// Mitsubishi GX Works2 project: group_35_Final   PLC: FX3G

// global labels: Global1
VAR_GLOBAL
  switch_check_start AT X007 : BOOL;
  cream AT D1100 : REAL;
END_VAR
VAR_GLOBAL CONSTANT
  con_false : BOOL := TRUE;
END_VAR
VAR_GLOBAL
  pulse_before_active AT X007 : BOOL;
  shity_pulse AT X011 : BOOL;
  chocolate AT D1200 : REAL;
END_VAR
VAR_GLOBAL CONSTANT
  con_chocolate : REAL := 240;
END_VAR
VAR_GLOBAL
  shity_pulse2 AT X007 : BOOL;
  shity_pulse1 AT X007 : BOOL;
  biscuit : BOOL;
END_VAR
VAR_GLOBAL CONSTANT
  con_biscuit : REAL := 6;
END_VAR
VAR_GLOBAL
  cream_input AT D1100 : REAL;
  lamp AT M2 : BOOL;
END_VAR
VAR_GLOBAL CONSTANT
  con300 : WORD := 400;
END_VAR
VAR_GLOBAL
  chocolate_input AT D1200 : REAL;
  biscit_inputnew AT D1300 : REAL;
END_VAR
VAR_GLOBAL CONSTANT
  constant6 : REAL := 6;
  contant240 : REAL := 240;
END_VAR
VAR_GLOBAL
  lamp_able_startDay AT Y002 : BOOL;
  ziluf_container : REAL;
  indicator_level1 AT Y001 : BOOL;
  kaki AT Y010 : BOOL;
  can_startday AT Y002 : BOOL;
  level1isgood AT Y001 : BOOL;
  level1done AT M2 : BOOL;
  zilufison AT X011 : BOOL;
  clockon AT TC0 : BOOL;
END_VAR
VAR_GLOBAL CONSTANT
  FourSec : REAL := 4;
  Fourcheck : WORD := 400;
END_VAR
VAR_GLOBAL
  Timer_Finish AT TS0 : BOOL;
  end_timer1 AT TS3 : BOOL;
  lamP1 AT Y005 : BOOL;
  Helo_Lamp AT M0 : BOOL;
END_VAR
VAR_GLOBAL CONSTANT
  Four_sec : INT := 40;
END_VAR
VAR_GLOBAL
  Timer_1 AT TC3 : BOOL;
END_VAR
VAR_GLOBAL CONSTANT
  One_sec : INT := 10;
END_VAR
VAR_GLOBAL
  Not_sufficnt_stuff AT M1 : BOOL;
  level1end AT Y006 : BOOL;
  lamp_2 AT Y001 : BOOL;
  Timer_2 AT TC4 : BOOL;
  TS300 : BOOL;
  end_Timer2 AT TS4 : BOOL;
  lamp_1 AT Y001 : BOOL;
  lamp0 AT Y000 : BOOL;
  Hiv_Huv_counter AT TC2 : BOOL;
  Hiv_Off AT TS2 : BOOL;
  lamp_10 AT Y001 : BOOL;
  lamp_6 AT Y006 : BOOL;
  lamp6 AT M6 : BOOL;
  Turn_on_mecA AT X010 : BOOL;
  plate_is_here AT X001 : BOOL;
  zilof_working AT Y004 : BOOL;
  high_sens AT X002 : BOOL;
  cam_sens AT X004 : BOOL;
  ziluf_lamp AT Y004 : BOOL;
  low_sens AT X003 : BOOL;
  biscuit_input : REAL;
END_VAR
VAR_GLOBAL CONSTANT
  con0 : REAL;
END_VAR
VAR_GLOBAL
  end_ziluf_lamp AT M12 : BOOL;
  qualtiy_check AT X006 : BOOL;
  analog_input AT D8280 : INT;
END_VAR
VAR_GLOBAL CONSTANT
  cons_400 : WORD := 400;
END_VAR
VAR_GLOBAL
  correct_analog AT D1111 : INT;
END_VAR
VAR_GLOBAL CONSTANT
  cons_5 : INT := 5;
END_VAR
VAR_GLOBAL
  what_is_it AT M12 : BOOL;
  yes AT M12 : BOOL;
  No AT M12 : BOOL;
END_VAR
VAR_GLOBAL CONSTANT
  cons_240 : REAL := 240;
END_VAR
VAR_GLOBAL
  con_chooclate : REAL;
END_VAR
VAR_GLOBAL CONSTANT
  cons_120 : REAL := 120;
  con400 : INT := 400;
  con300ww : REAL := 300;
END_VAR
VAR_GLOBAL
  Tvila_container : REAL;
  Tvila_timmer AT TC5 : BOOL;
END_VAR
VAR_GLOBAL CONSTANT
  tree_sec : INT := 50;
END_VAR
VAR_GLOBAL
  stop_tvila AT TS5 : BOOL;
  lamp3_off AT Y003 : BOOL;
END_VAR
VAR_GLOBAL CONSTANT
  Five_sec : INT := 50;
END_VAR
VAR_GLOBAL
  dayison AT Y007 : BOOL;
  day_is_on AT M0 : BOOL;
  lamp7 AT Y007 : BOOL;
  finish_packing AT Y002 : BOOL;
  switch_x0 AT X000 : BOOL;
  cc0_press5 AT CC0 : BOOL;
END_VAR
VAR_GLOBAL CONSTANT
  count_5 : WORD := K5;
END_VAR
VAR_GLOBAL
  switch_end_count AT CS13 : BOOL;
  m2_stop_light AT Y002 : BOOL;
  Reset_count AT Y002 : BOOL;
  Light_Y2 AT Y002 : BOOL;
  Fin6 AT Y002 : BOOL;
  Finished AT D1400 : REAL;
  count_6 AT K6 : INT;
  Stored AT D1400 : INT;
END_VAR
VAR_GLOBAL CONSTANT
  const_6 : REAL := 40;
END_VAR
VAR_GLOBAL
  Ana_Dozens AT D8282 : INT;
  ValueForOutput : REAL;
  analog_ouput AT D8282 : REAL;
  analog_output82 AT D8282 : INT;
  HELP_OUTPUT AT Y011 : BOOL;
  M_11 AT M11 : BOOL;
END_VAR
VAR_GLOBAL CONSTANT
  con_crembo6 : REAL := 6;
END_VAR
VAR_GLOBAL
  HELP_lamp_endPack AT M11 : BOOL;
END_VAR
VAR_GLOBAL CONSTANT
  con_40 : REAL := 40;
END_VAR
VAR_GLOBAL
  help_end_output AT M12 : BOOL;
  Finished_crembo AT D4000 : REAL;
  M23_finishedCH AT M23 : BOOL;
  CC13_press6 AT CC13 : BOOL;
  coub AT K6 : INT;
  M21_finish6 AT M21 : BOOL;
  press_5_finish AT CS0 : BOOL;
  press6_finished AT CS13 : BOOL;
  Restarter AT CC0 : BOOL;
  Restarter13 AT CC13 : BOOL;
  CC10_press6 AT CC10 : BOOL;
  reset0 AT CC0 : BOOL;
  reset13 AT CC13 : BOOL;
  finish_creambo AT CS13 : BOOL;
  Push_to_Spray AT X005 : BOOL;
  Sen_Full AT X004 : BOOL;
  Sen_plate AT X003 : BOOL;
  Spray AT TC6 : BOOL;
END_VAR
VAR_GLOBAL CONSTANT
  count_5sec : INT := K50;
END_VAR
VAR_GLOBAL
  Spray_light AT Y000 : BOOL;
  Spray_Timer AT TS6 : BOOL;
  HelpNOGelem AT M34 : BOOL;
  TimerEndDay AT TC9 : BOOL;
  EndDay3min AT K30 : INT;
  stop_blinking AT TS57 : BOOL;
  HELP_lamp_endday AT M5 : BOOL;
  yesGelem AT M19 : BOOL;
  finishGelem AT Y002 : BOOL;
  finishGelemCounter AT CC6 : BOOL;
END_VAR
VAR_GLOBAL CONSTANT
  count_6_finish : INT := 6;
END_VAR
VAR_GLOBAL
  finish_itertion AT Y002 : BOOL;
END_VAR
VAR_GLOBAL CONSTANT
  EndDay3sec : INT := 30;
END_VAR
VAR_GLOBAL
  TS_57 AT TS57 : BOOL;
  lamp_blinking1 AT M2 : BOOL;
  stop_blink_lamp AT M8 : BOOL;
  lamp_blinking2 AT M9 : BOOL;
  TS_7 AT TS7 : BOOL;
  TC_7 AT TS7 : BOOL;
  TC_8 AT TC8 : BOOL;
  TS_8 AT TS8 : BOOL;
  lamp_timer AT TC8 : BOOL;
  lamp_timer7 AT TC7 : BOOL;
  lamp_timer8 AT TC8 : BOOL;
  lt8 AT TS8 : BOOL;
  lt_7 AT TS7 : BOOL;
  end_lamp AT TS9 : BOOL;
  chocolate_container AT D1201 : REAL;
  biscuit_container AT D1301 : REAL;
  cream_container AT D1101 : REAL;
  Shut_Down_ziluf AT X005 : BOOL;
  Next_phase3 AT M12 : BOOL;
  lamp12 AT M120 : BOOL;
  Next_phase4 AT M120 : BOOL;
END_VAR

// task Task_01 (event TRUE, interval 0, priority 31): POU_01

PROGRAM POU_01
VAR CONSTANT
  con_cream : REAL := 300;
  con6 : REAL := 6;
END_VAR
VAR
  TC100 : BOOL;
  cam : BOOL;
END_VAR
(* structured ladder/FBD written out as ST: instructions are called as NAME(EN, inputs, outputs); _pN, _eN, _tN stand for wires *)
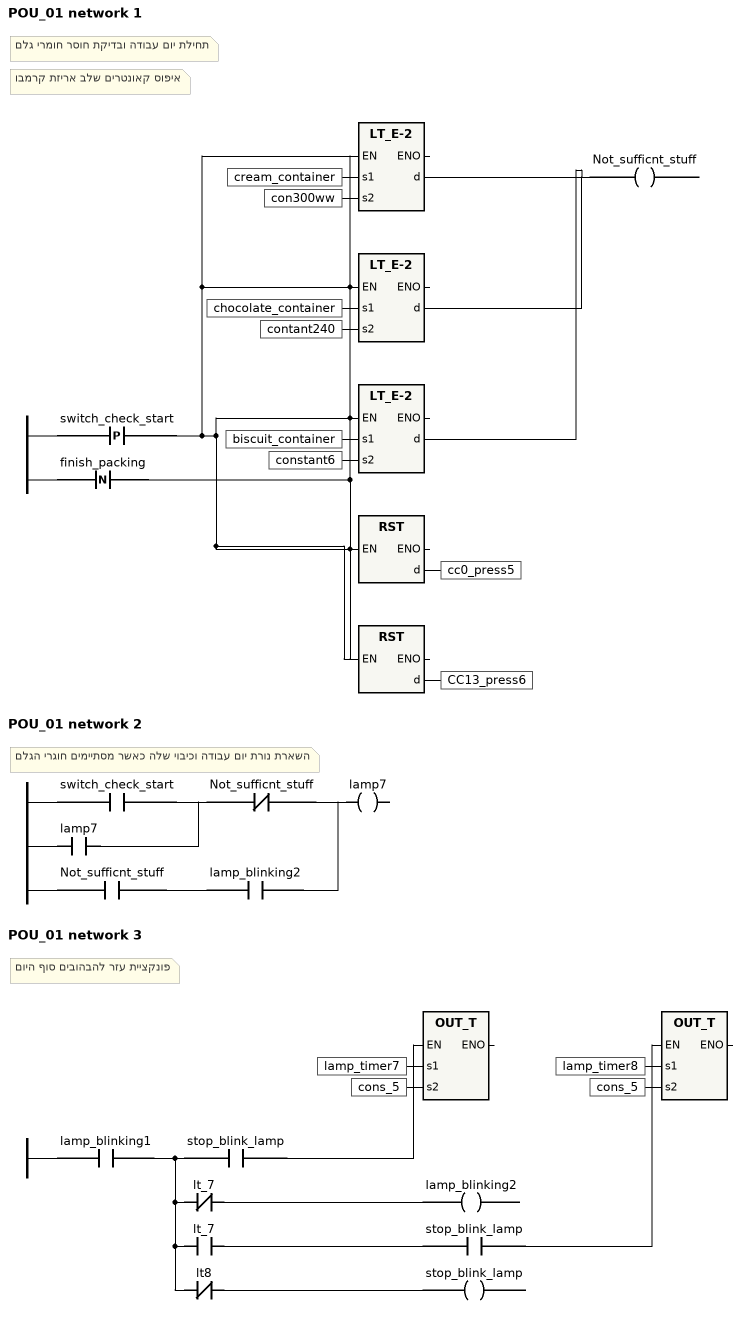
(* network 1 *)
(* תחילת יום עבודה ובדיקת חוסר חומרי גלם *)
(* איפוס קאונטרים שלב אריזת קרמבו *)
_p1 := LDP(TRUE, switch_check_start) OR LDF(TRUE, finish_packing);
LT_E(_p1, cream_container, con300ww, _t2);
LT_E(_p1, chocolate_container, contant240, _t3);
LT_E(_p1, biscuit_container, constant6, _t4);
Not_sufficnt_stuff := _t2 OR _t3 OR _t4;
RST(_p1, cc0_press5);
RST(_p1, CC13_press6);
(* network 2 *)
(* השארת נורת יום עבודה וכיבוי שלה כאשר מסתיימים חוגרי הגלם *)
lamp7 := ((switch_check_start OR lamp7) AND NOT Not_sufficnt_stuff) OR (Not_sufficnt_stuff AND lamp_blinking2);
(* network 3 *)
(* פונקציית עזר להבהובים סוף היום *)
OUT_T(lamp_blinking1 AND stop_blink_lamp, lamp_timer7, cons_5);
lamp_blinking2 := lamp_blinking1 AND NOT lt_7;
OUT_T(lamp_blinking1 AND lt_7 AND stop_blink_lamp, lamp_timer8, cons_5);
stop_blink_lamp := lamp_blinking1 AND NOT lt8;
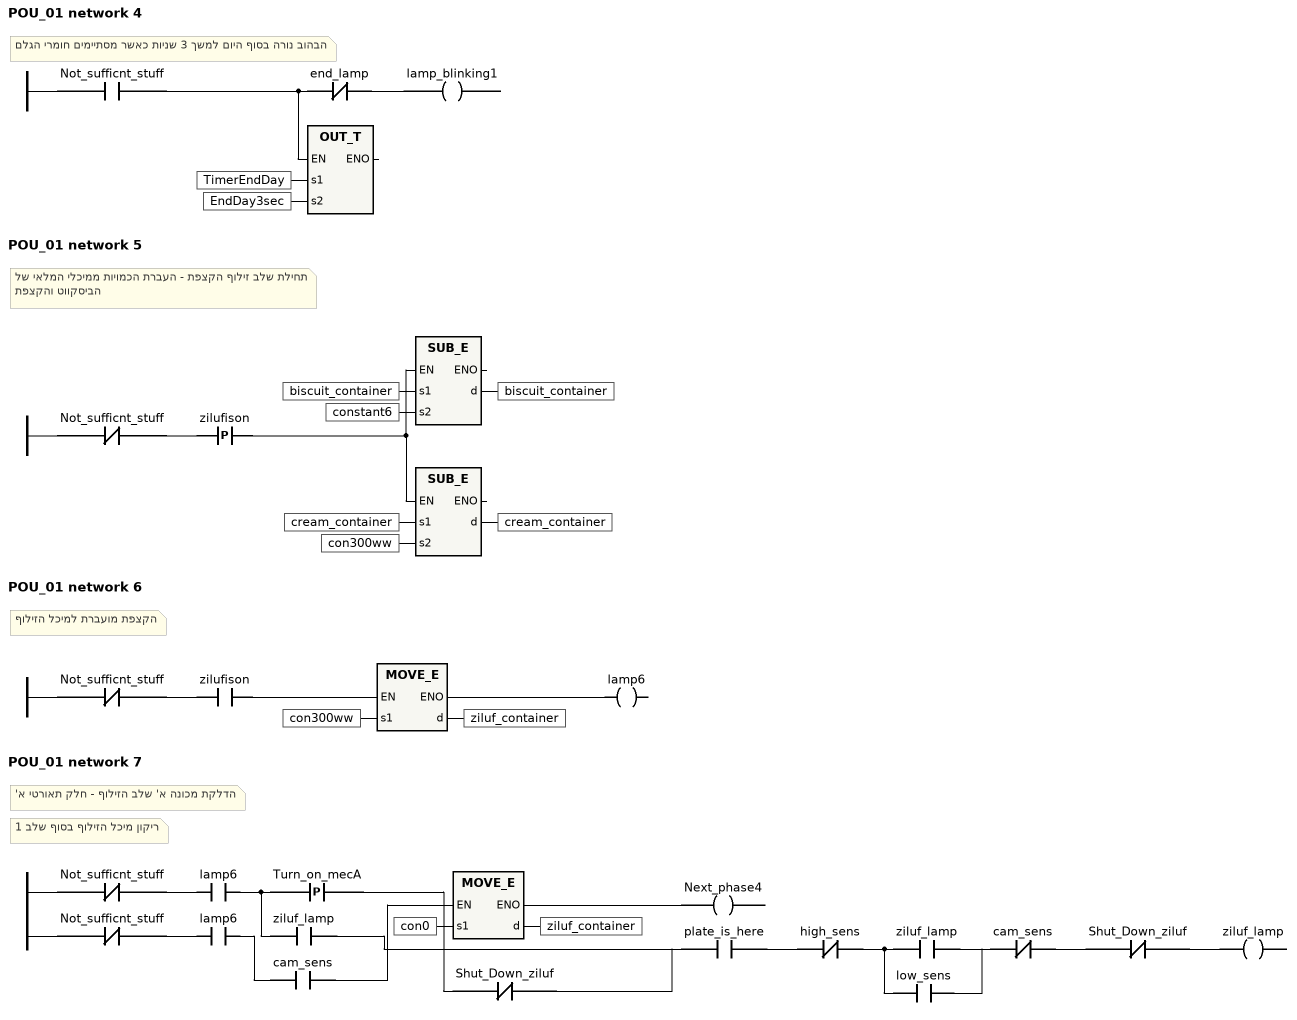
(* network 4 *)
(* הבהוב נורה בסוף היום למשך 3 שניות כאשר מסתיימים חומרי הגלם *)
lamp_blinking1 := Not_sufficnt_stuff AND NOT end_lamp;
OUT_T(Not_sufficnt_stuff, TimerEndDay, EndDay3sec);
(* network 5 *)
(* תחילת שלב זילוף הקצפת - העברת הכמויות ממיכלי המלאי של הביסקווט והקצפת *)
_p1 := NOT Not_sufficnt_stuff AND LDP(TRUE, zilufison);
SUB_E(_p1, biscuit_container, constant6, biscuit_container);
SUB_E(_p1, cream_container, con300ww, cream_container);
(* network 6 *)
(* הקצפת מועברת למיכל הזילוף *)
_e1 := MOVE_E(NOT Not_sufficnt_stuff AND zilufison, con300ww, ziluf_container);
lamp6 := _e1;
(* network 7 *)
(* הדלקת מכונה א' שלב הזילוף - חלק תאורטי א' *)
(* ריקון מיכל הזילוף בסוף שלב 1 *)
_p1 := NOT Not_sufficnt_stuff AND lamp6;
_p2 := (((_p1 AND LDP(TRUE, Turn_on_mecA) AND NOT Shut_Down_ziluf) OR (_p1 AND ziluf_lamp)) AND plate_is_here) AND NOT high_sens;
ziluf_lamp := (((_p2 AND ziluf_lamp) OR (_p2 AND low_sens)) AND NOT cam_sens) AND NOT Shut_Down_ziluf;
_e3 := MOVE_E(NOT Not_sufficnt_stuff AND lamp6 AND cam_sens, con0, ziluf_container);
Next_phase4 := _e3;
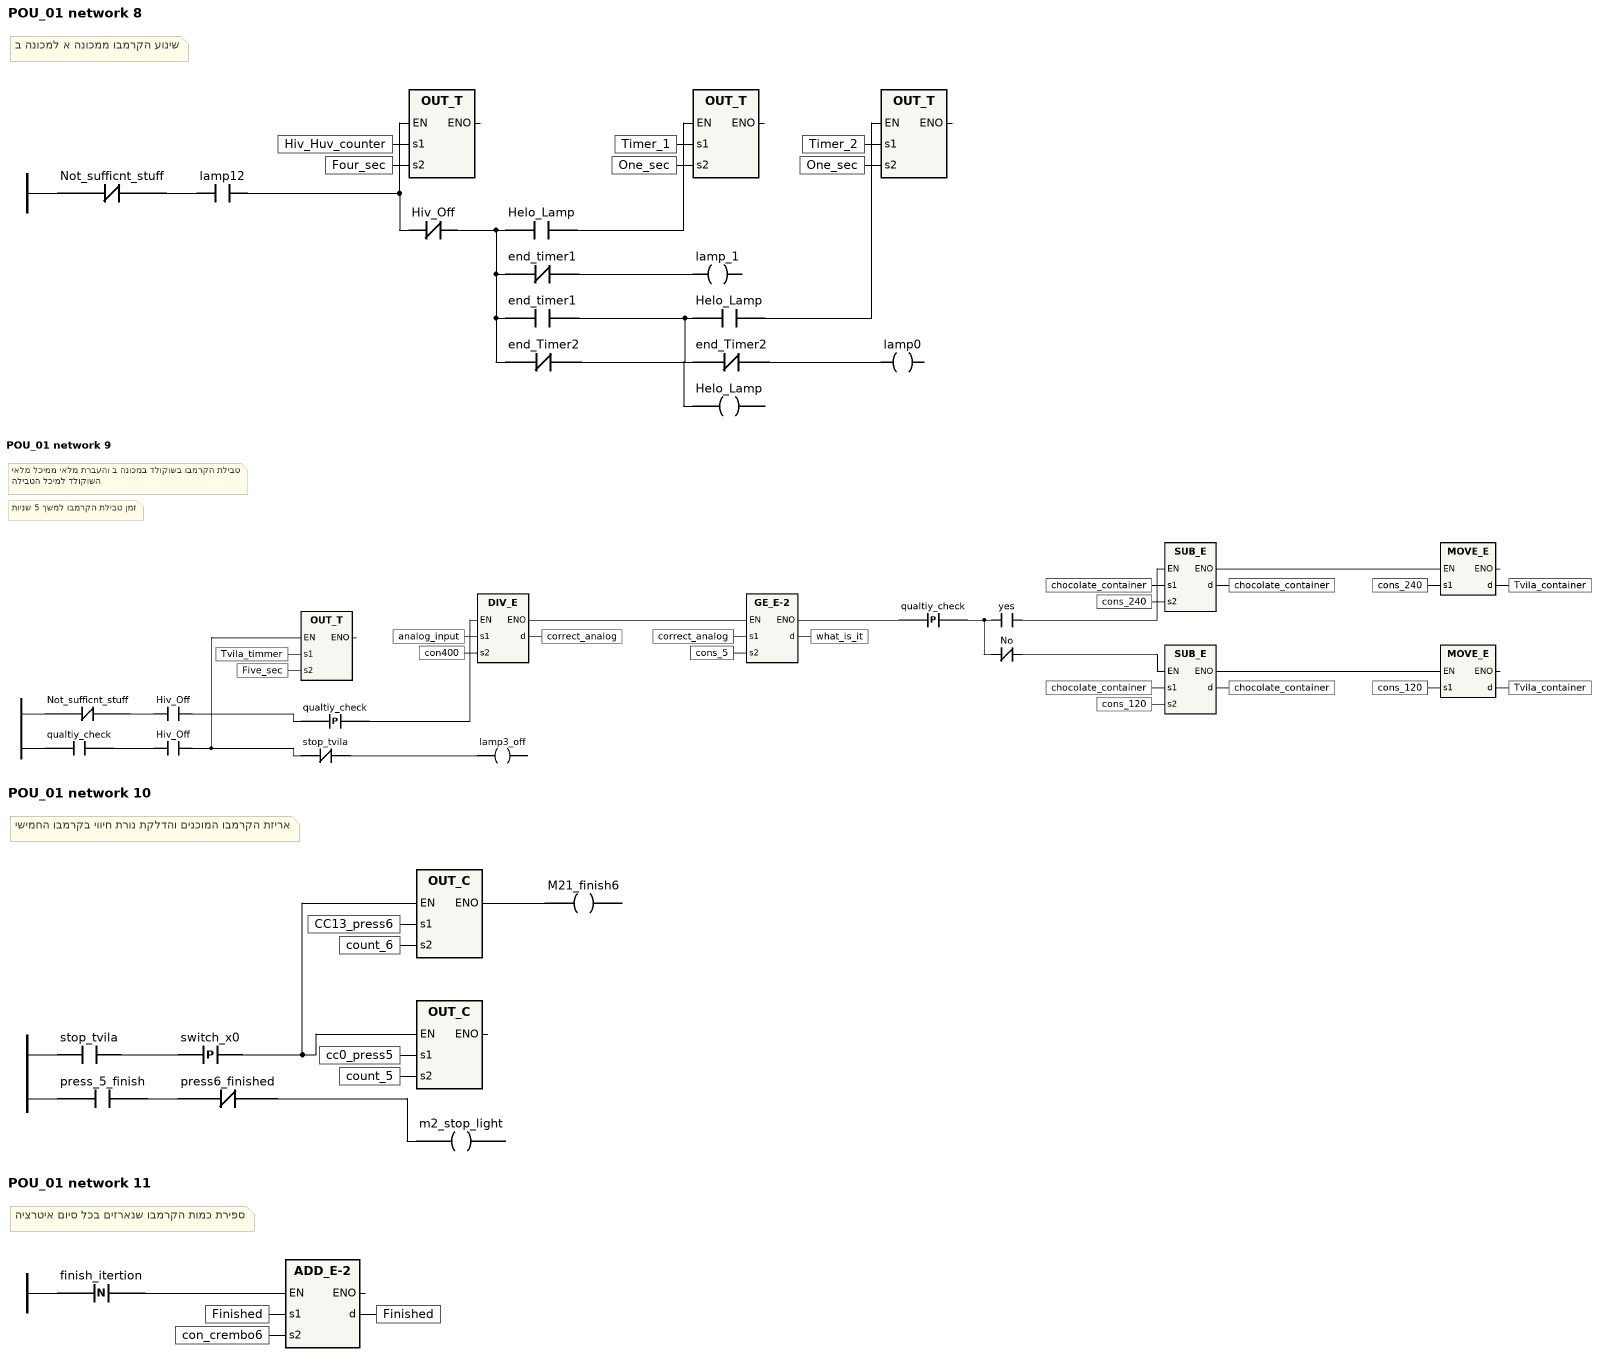
(* network 8 *)
(* שינוע הקרמבו ממכונה א למכונה ב *)
_p1 := NOT Not_sufficnt_stuff AND lamp12;
OUT_T(_p1, Hiv_Huv_counter, Four_sec);
_p2 := _p1 AND NOT Hiv_Off;
OUT_T(_p2 AND Helo_Lamp, Timer_1, One_sec);
lamp_1 := _p2 AND NOT end_timer1;
_p3 := _p2 AND end_timer1;
OUT_T(_p3 AND Helo_Lamp, Timer_2, One_sec);
lamp0 := _p3 AND NOT end_Timer2;
Helo_Lamp := _p2 AND NOT end_Timer2;
(* network 9 *)
(* טבילת הקרמבו בשוקולד במכונה ב והעברת מלאי ממיכל מלאי השוקולד למיכל הטבילה *)
(* זמן טבילת הקרמבו למשך 5 שניות *)
_e1 := DIV_E(NOT Not_sufficnt_stuff AND Hiv_Off AND LDP(TRUE, qualtiy_check), analog_input, con400, correct_analog);
_e2 := GE_E(_e1, correct_analog, cons_5, what_is_it);
_p3 := _e2 AND LDP(TRUE, qualtiy_check);
_e4 := SUB_E(_p3 AND yes, chocolate_container, cons_240, chocolate_container);
MOVE_E(_e4, cons_240, Tvila_container);
_e5 := SUB_E(_p3 AND NOT No, chocolate_container, cons_120, chocolate_container);
MOVE_E(_e5, cons_120, Tvila_container);
_p6 := qualtiy_check AND Hiv_Off;
lamp3_off := _p6 AND NOT stop_tvila;
OUT_T(_p6, Tvila_timmer, Five_sec);
(* network 10 *)
(* אריזת הקרמבו המוכנים והדלקת נורת חיווי בקרמבו החמישי *)
_p1 := stop_tvila AND LDP(TRUE, switch_x0);
OUT_C(_p1, cc0_press5, count_5);
_e2 := OUT_C(_p1, CC13_press6, count_6);
M21_finish6 := _e2;
m2_stop_light := press_5_finish AND NOT press6_finished;
(* network 11 *)
(* ספירת כמות הקרמבו שנארזים בכל סיום איטרציה *)
ADD_E(LDF(TRUE, finish_itertion), Finished, con_crembo6, Finished);
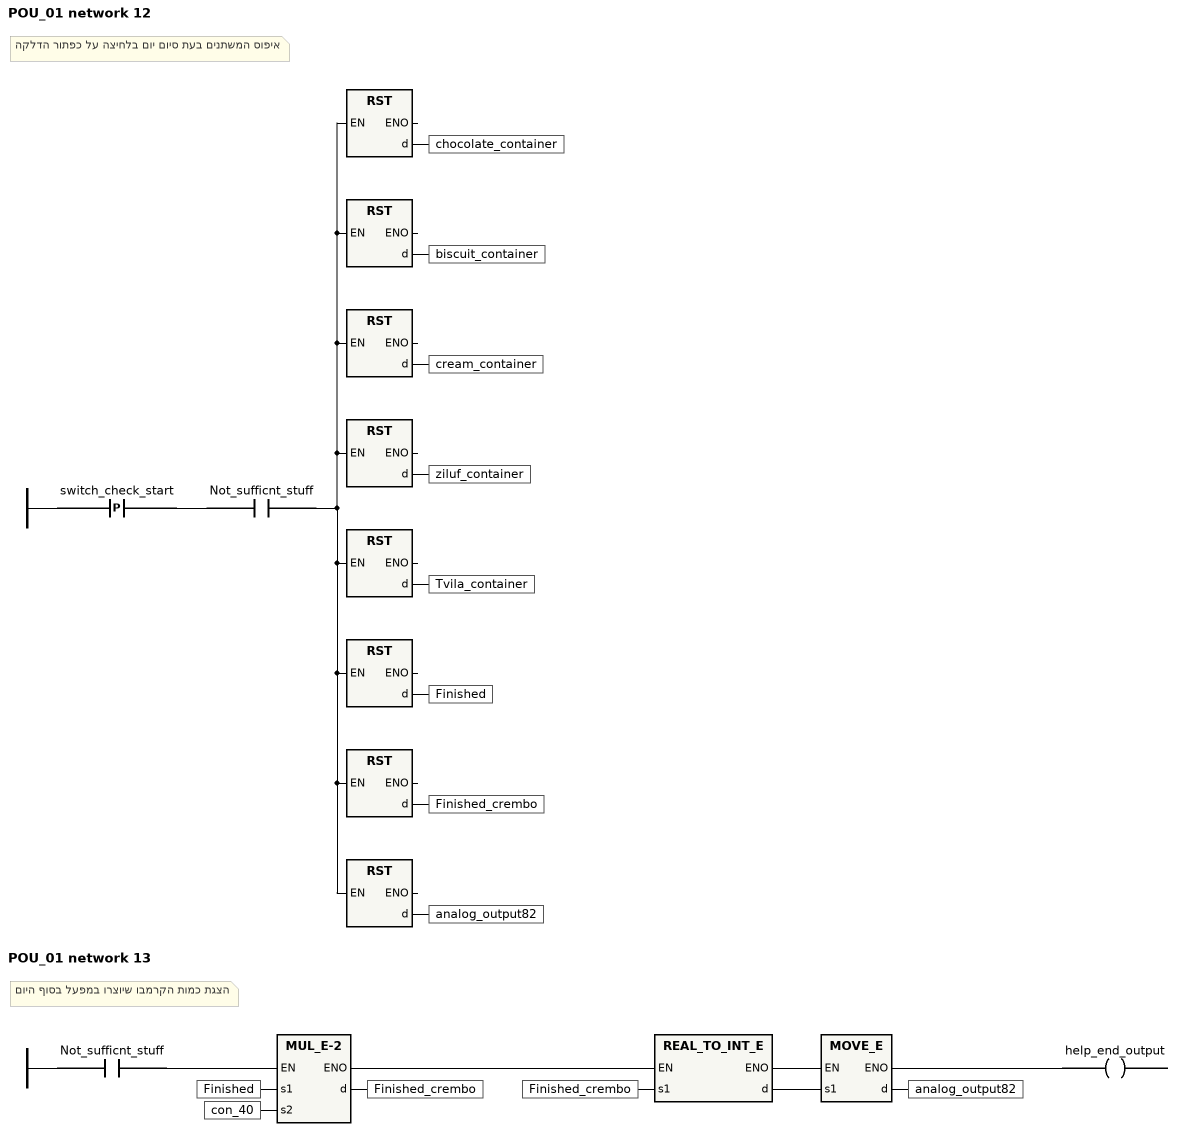
(* network 12 *)
(* איפוס המשתנים בעת סיום יום בלחיצה על כפתור הדלקה *)
_p1 := LDP(TRUE, switch_check_start) AND Not_sufficnt_stuff;
RST(_p1, chocolate_container);
RST(_p1, biscuit_container);
RST(_p1, cream_container);
RST(_p1, ziluf_container);
RST(_p1, Tvila_container);
RST(_p1, Finished);
RST(_p1, Finished_crembo);
RST(_p1, analog_output82);
(* network 13 *)
(* הצגת כמות הקרמבו שיוצרו במפעל בסוף היום *)
_e1 := MUL_E(Not_sufficnt_stuff, Finished, con_40, Finished_crembo);
_e3 := REAL_TO_INT_E(_e1, Finished_crembo, _t2);
_e4 := MOVE_E(_e3, _t2, analog_output82);
help_end_output := _e4;
END_PROGRAM
